PROGRAM JIG_PARTPRESENT
VAR
END_VAR

END_PROGRAM

(* stored: Version 1.1.0.1, ProductVersion 3.1.4022.18
   POU JIG_PARTPRESENT: Id {1d54f2cf-eae3-4146-b82e-ed6373ce7f4a}, SpecialFunc None *)
